# EPICS autosave request: iocBoot/generic_motors_ioc/dbSave/KB_Hz_.req
%
% BURT Request File
%
% $(P)KB:Hz:  Horizontal KB mirror Z-positioning
%

file assy.req ASSY=$(P)KB:Hz
$(P)KB:Hz:Base1:23
$(P)KB:Hz:Base23
file mtr1.req MTR1=$(P)KB:mhz1
file mtr1.req MTR1=$(P)KB:mhz2
file mtr1.req MTR1=$(P)KB:mhz3
file drv1.req DRV1=$(P)KB:HZ1
file drv1.req DRV1=$(P)KB:HZ2
file drv1.req DRV1=$(P)KB:HZ3
file axs1.req AXS1=$(P)KB:HL
file axs1.req AXS1=$(P)KB:HW
file axs1.req AXS1=$(P)KB:HR
